Staubli VAL3: SerialPort.pjx

Parameters version=s7.9 stackSize=5000 millimeterUnit=true
Program file=start.pgx
Program file=stop.pgx
Data file=SerialPort.dtx
